Xinje XDPPro project, PLC1: XDM-60T10 (software 3.5.3 2018-12-07)

PROGRAM Ladder

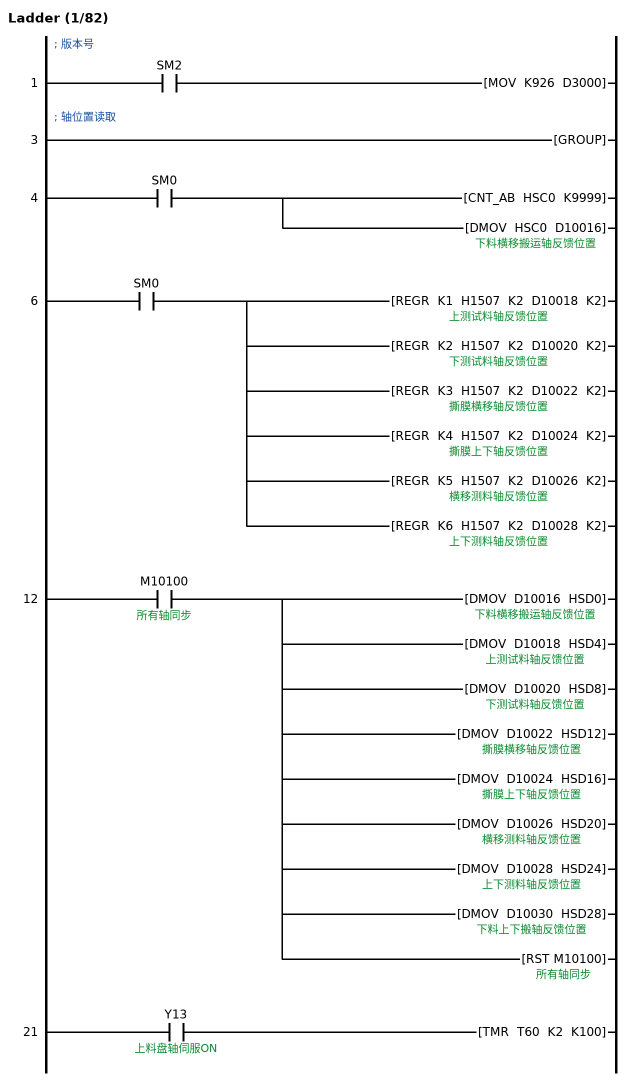
; 版本号
LD     SM2
MOV    K926 D3000
; 轴位置读取
GROUP
LD     SM0
CNT_AB HSC0 K9999
DMOV   HSC0 D10016	; 下料横移搬运轴反馈位置
LD     SM0
REGR   K1 H1507 K2 D10018 K2	; 上测试料轴反馈位置
REGR   K2 H1507 K2 D10020 K2	; 下测试料轴反馈位置
REGR   K3 H1507 K2 D10022 K2	; 撕膜横移轴反馈位置
REGR   K4 H1507 K2 D10024 K2	; 撕膜上下轴反馈位置
REGR   K5 H1507 K2 D10026 K2	; 横移测料轴反馈位置
REGR   K6 H1507 K2 D10028 K2	; 上下测料轴反馈位置
LD     M10100	; 所有轴同步
DMOV   D10016 HSD0	; 下料横移搬运轴反馈位置
DMOV   D10018 HSD4	; 上测试料轴反馈位置
DMOV   D10020 HSD8	; 下测试料轴反馈位置
DMOV   D10022 HSD12	; 撕膜横移轴反馈位置
DMOV   D10024 HSD16	; 撕膜上下轴反馈位置
DMOV   D10026 HSD20	; 横移测料轴反馈位置
DMOV   D10028 HSD24	; 上下测料轴反馈位置
DMOV   D10030 HSD28	; 下料上下搬轴反馈位置
RST    M10100	; 所有轴同步
LD     Y13	; 上料盘轴伺服ON
TMR    T60 K2 K100

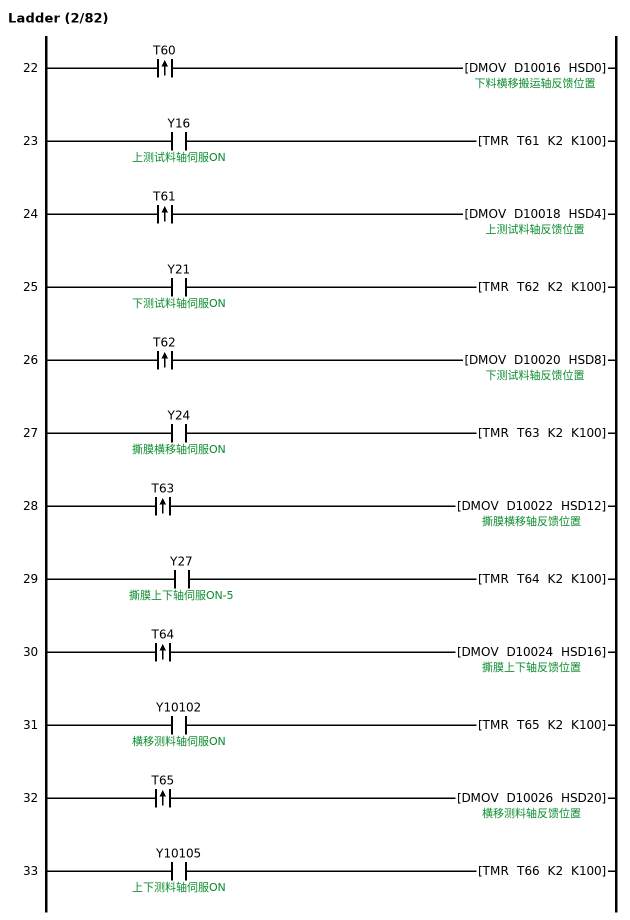
LDP    T60
DMOV   D10016 HSD0	; 下料横移搬运轴反馈位置
LD     Y16	; 上测试料轴伺服ON
TMR    T61 K2 K100
LDP    T61
DMOV   D10018 HSD4	; 上测试料轴反馈位置
LD     Y21	; 下测试料轴伺服ON
TMR    T62 K2 K100
LDP    T62
DMOV   D10020 HSD8	; 下测试料轴反馈位置
LD     Y24	; 撕膜横移轴伺服ON
TMR    T63 K2 K100
LDP    T63
DMOV   D10022 HSD12	; 撕膜横移轴反馈位置
LD     Y27	; 撕膜上下轴伺服ON-5
TMR    T64 K2 K100
LDP    T64
DMOV   D10024 HSD16	; 撕膜上下轴反馈位置
LD     Y10102	; 横移测料轴伺服ON
TMR    T65 K2 K100
LDP    T65
DMOV   D10026 HSD20	; 横移测料轴反馈位置
LD     Y10105	; 上下测料轴伺服ON
TMR    T66 K2 K100

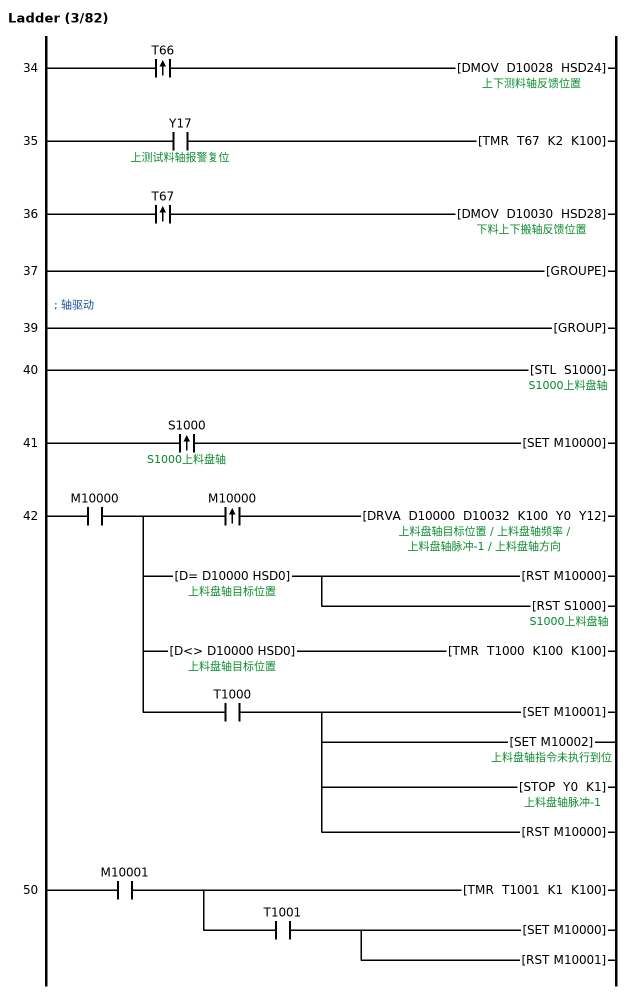
LDP    T66
DMOV   D10028 HSD24	; 上下测料轴反馈位置
LD     Y17	; 上测试料轴报警复位
TMR    T67 K2 K100
LDP    T67
DMOV   D10030 HSD28	; 下料上下搬轴反馈位置
GROUPE
; 轴驱动
GROUP
STL    S1000	; S1000上料盘轴
LDP    S1000	; S1000上料盘轴
SET    M10000
LD     M10000
MPS
ANDP   M10000
DRVA   D10000 D10032 K100 Y0 Y12	; 上料盘轴目标位置 / 上料盘轴频率 / 上料盘轴脉冲-1 / 上料盘轴方向
MRD
DAND=  D10000 HSD0	; 上料盘轴目标位置
RST    M10000
RST    S1000	; S1000上料盘轴
MRD
DAND<> D10000 HSD0	; 上料盘轴目标位置
TMR    T1000 K100 K100
MPP
AND    T1000
SET    M10001
SET    M10002	; 上料盘轴指令未执行到位
STOP   Y0 K1	; 上料盘轴脉冲-1
RST    M10000
LD     M10001
TMR    T1001 K1 K100
AND    T1001
SET    M10000
RST    M10001

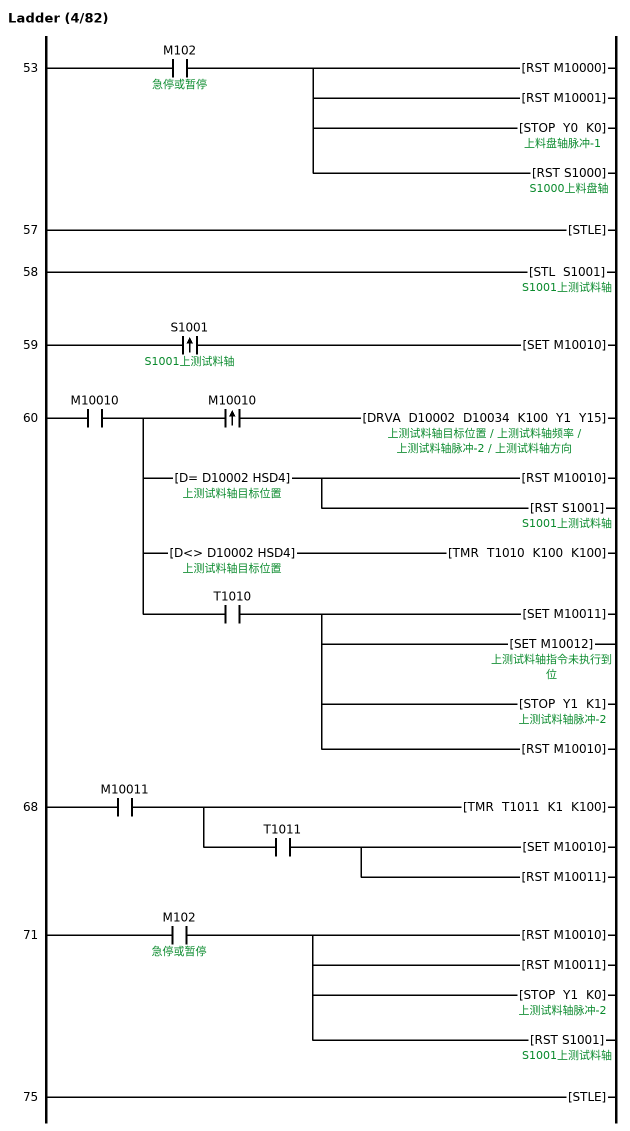
LD     M102	; 急停或暂停
RST    M10000
RST    M10001
STOP   Y0 K0	; 上料盘轴脉冲-1
RST    S1000	; S1000上料盘轴
STLE
STL    S1001	; S1001上测试料轴
LDP    S1001	; S1001上测试料轴
SET    M10010
LD     M10010
MPS
ANDP   M10010
DRVA   D10002 D10034 K100 Y1 Y15	; 上测试料轴目标位置 / 上测试料轴频率 / 上测试料轴脉冲-2 / 上测试料轴方向
MRD
DAND=  D10002 HSD4	; 上测试料轴目标位置
RST    M10010
RST    S1001	; S1001上测试料轴
MRD
DAND<> D10002 HSD4	; 上测试料轴目标位置
TMR    T1010 K100 K100
MPP
AND    T1010
SET    M10011
SET    M10012	; 上测试料轴指令未执行到位
STOP   Y1 K1	; 上测试料轴脉冲-2
RST    M10010
LD     M10011
TMR    T1011 K1 K100
AND    T1011
SET    M10010
RST    M10011
LD     M102	; 急停或暂停
RST    M10010
RST    M10011
STOP   Y1 K0	; 上测试料轴脉冲-2
RST    S1001	; S1001上测试料轴
STLE

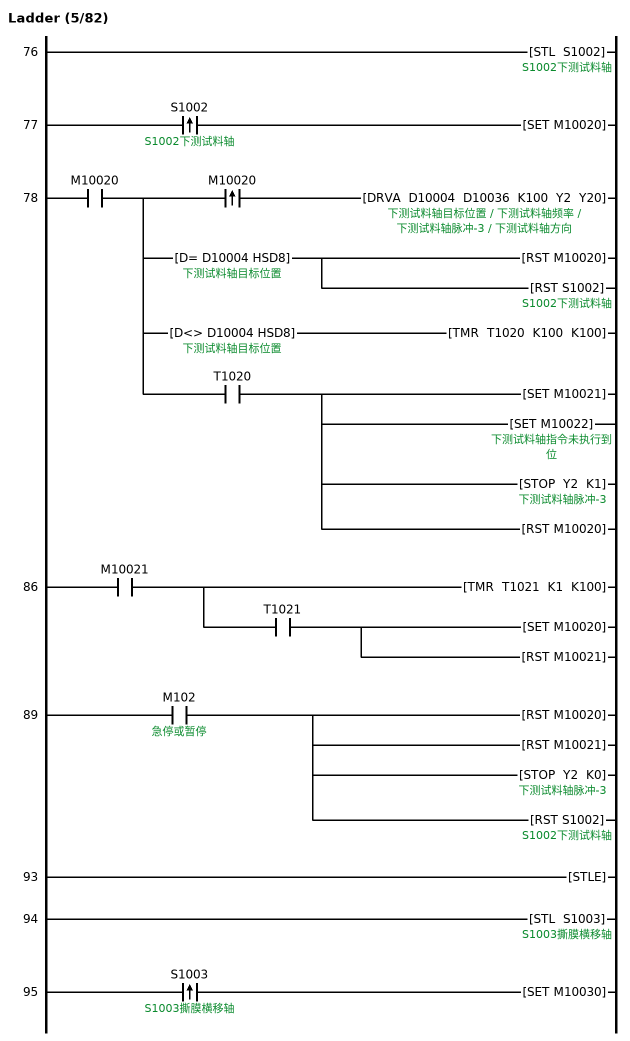
STL    S1002	; S1002下测试料轴
LDP    S1002	; S1002下测试料轴
SET    M10020
LD     M10020
MPS
ANDP   M10020
DRVA   D10004 D10036 K100 Y2 Y20	; 下测试料轴目标位置 / 下测试料轴频率 / 下测试料轴脉冲-3 / 下测试料轴方向
MRD
DAND=  D10004 HSD8	; 下测试料轴目标位置
RST    M10020
RST    S1002	; S1002下测试料轴
MRD
DAND<> D10004 HSD8	; 下测试料轴目标位置
TMR    T1020 K100 K100
MPP
AND    T1020
SET    M10021
SET    M10022	; 下测试料轴指令未执行到位
STOP   Y2 K1	; 下测试料轴脉冲-3
RST    M10020
LD     M10021
TMR    T1021 K1 K100
AND    T1021
SET    M10020
RST    M10021
LD     M102	; 急停或暂停
RST    M10020
RST    M10021
STOP   Y2 K0	; 下测试料轴脉冲-3
RST    S1002	; S1002下测试料轴
STLE
STL    S1003	; S1003撕膜横移轴
LDP    S1003	; S1003撕膜横移轴
SET    M10030

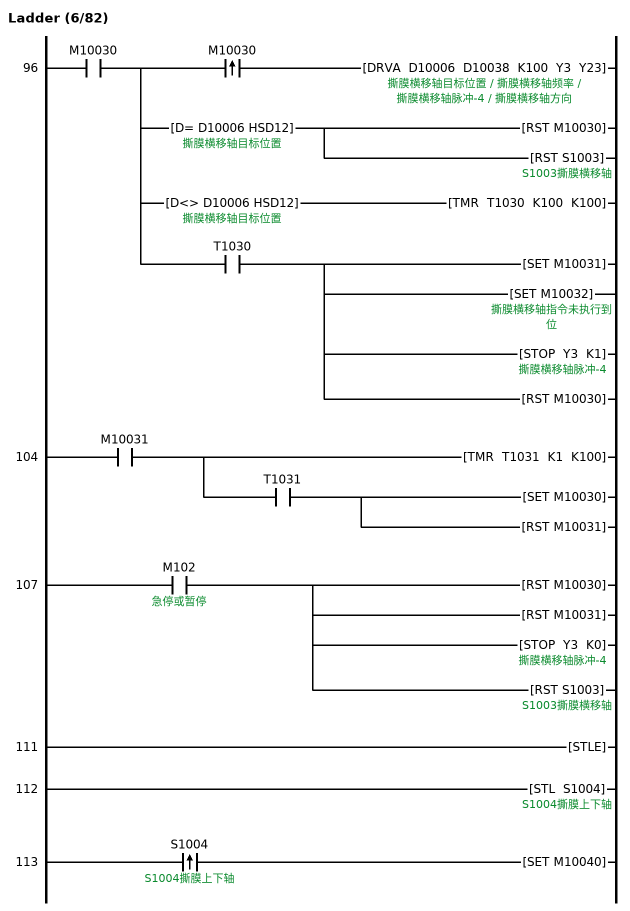
LD     M10030
MPS
ANDP   M10030
DRVA   D10006 D10038 K100 Y3 Y23	; 撕膜横移轴目标位置 / 撕膜横移轴频率 / 撕膜横移轴脉冲-4 / 撕膜横移轴方向
MRD
DAND=  D10006 HSD12	; 撕膜横移轴目标位置
RST    M10030
RST    S1003	; S1003撕膜横移轴
MRD
DAND<> D10006 HSD12	; 撕膜横移轴目标位置
TMR    T1030 K100 K100
MPP
AND    T1030
SET    M10031
SET    M10032	; 撕膜横移轴指令未执行到位
STOP   Y3 K1	; 撕膜横移轴脉冲-4
RST    M10030
LD     M10031
TMR    T1031 K1 K100
AND    T1031
SET    M10030
RST    M10031
LD     M102	; 急停或暂停
RST    M10030
RST    M10031
STOP   Y3 K0	; 撕膜横移轴脉冲-4
RST    S1003	; S1003撕膜横移轴
STLE
STL    S1004	; S1004撕膜上下轴
LDP    S1004	; S1004撕膜上下轴
SET    M10040

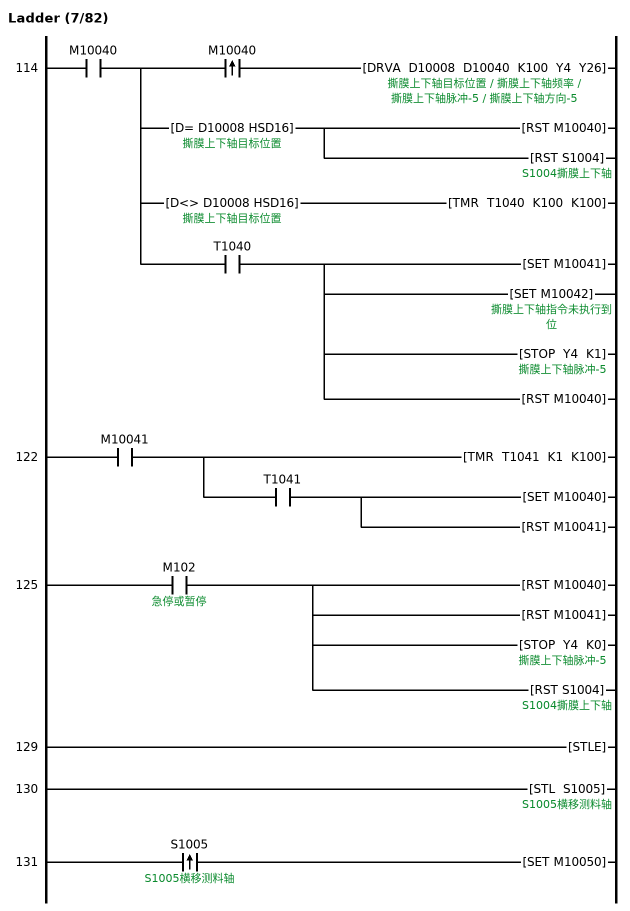
LD     M10040
MPS
ANDP   M10040
DRVA   D10008 D10040 K100 Y4 Y26	; 撕膜上下轴目标位置 / 撕膜上下轴频率 / 撕膜上下轴脉冲-5 / 撕膜上下轴方向-5
MRD
DAND=  D10008 HSD16	; 撕膜上下轴目标位置
RST    M10040
RST    S1004	; S1004撕膜上下轴
MRD
DAND<> D10008 HSD16	; 撕膜上下轴目标位置
TMR    T1040 K100 K100
MPP
AND    T1040
SET    M10041
SET    M10042	; 撕膜上下轴指令未执行到位
STOP   Y4 K1	; 撕膜上下轴脉冲-5
RST    M10040
LD     M10041
TMR    T1041 K1 K100
AND    T1041
SET    M10040
RST    M10041
LD     M102	; 急停或暂停
RST    M10040
RST    M10041
STOP   Y4 K0	; 撕膜上下轴脉冲-5
RST    S1004	; S1004撕膜上下轴
STLE
STL    S1005	; S1005横移测料轴
LDP    S1005	; S1005横移测料轴
SET    M10050

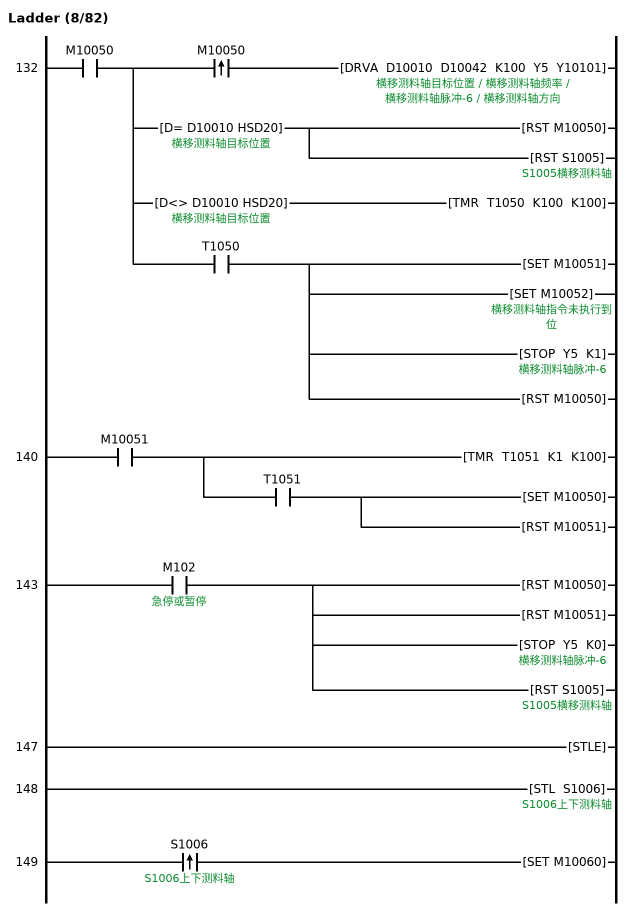
LD     M10050
MPS
ANDP   M10050
DRVA   D10010 D10042 K100 Y5 Y10101	; 横移测料轴目标位置 / 横移测料轴频率 / 横移测料轴脉冲-6 / 横移测料轴方向
MRD
DAND=  D10010 HSD20	; 横移测料轴目标位置
RST    M10050
RST    S1005	; S1005横移测料轴
MRD
DAND<> D10010 HSD20	; 横移测料轴目标位置
TMR    T1050 K100 K100
MPP
AND    T1050
SET    M10051
SET    M10052	; 横移测料轴指令未执行到位
STOP   Y5 K1	; 横移测料轴脉冲-6
RST    M10050
LD     M10051
TMR    T1051 K1 K100
AND    T1051
SET    M10050
RST    M10051
LD     M102	; 急停或暂停
RST    M10050
RST    M10051
STOP   Y5 K0	; 横移测料轴脉冲-6
RST    S1005	; S1005横移测料轴
STLE
STL    S1006	; S1006上下测料轴
LDP    S1006	; S1006上下测料轴
SET    M10060

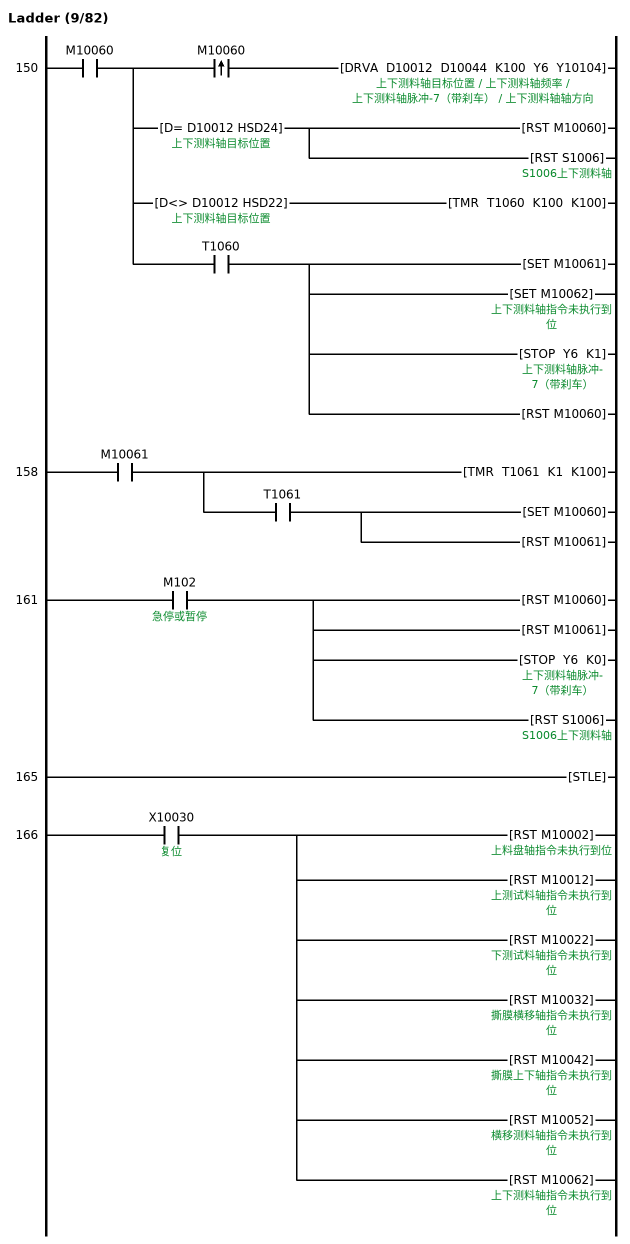
LD     M10060
MPS
ANDP   M10060
DRVA   D10012 D10044 K100 Y6 Y10104	; 上下测料轴目标位置 / 上下测料轴频率 / 上下测料轴脉冲-7（带刹车） / 上下测料轴轴方向
MRD
DAND=  D10012 HSD24	; 上下测料轴目标位置
RST    M10060
RST    S1006	; S1006上下测料轴
MRD
DAND<> D10012 HSD22	; 上下测料轴目标位置
TMR    T1060 K100 K100
MPP
AND    T1060
SET    M10061
SET    M10062	; 上下测料轴指令未执行到位
STOP   Y6 K1	; 上下测料轴脉冲-7（带刹车）
RST    M10060
LD     M10061
TMR    T1061 K1 K100
AND    T1061
SET    M10060
RST    M10061
LD     M102	; 急停或暂停
RST    M10060
RST    M10061
STOP   Y6 K0	; 上下测料轴脉冲-7（带刹车）
RST    S1006	; S1006上下测料轴
STLE
LD     X10030	; 复位
RST    M10002	; 上料盘轴指令未执行到位
RST    M10012	; 上测试料轴指令未执行到位
RST    M10022	; 下测试料轴指令未执行到位
RST    M10032	; 撕膜横移轴指令未执行到位
RST    M10042	; 撕膜上下轴指令未执行到位
RST    M10052	; 横移测料轴指令未执行到位
RST    M10062	; 上下测料轴指令未执行到位

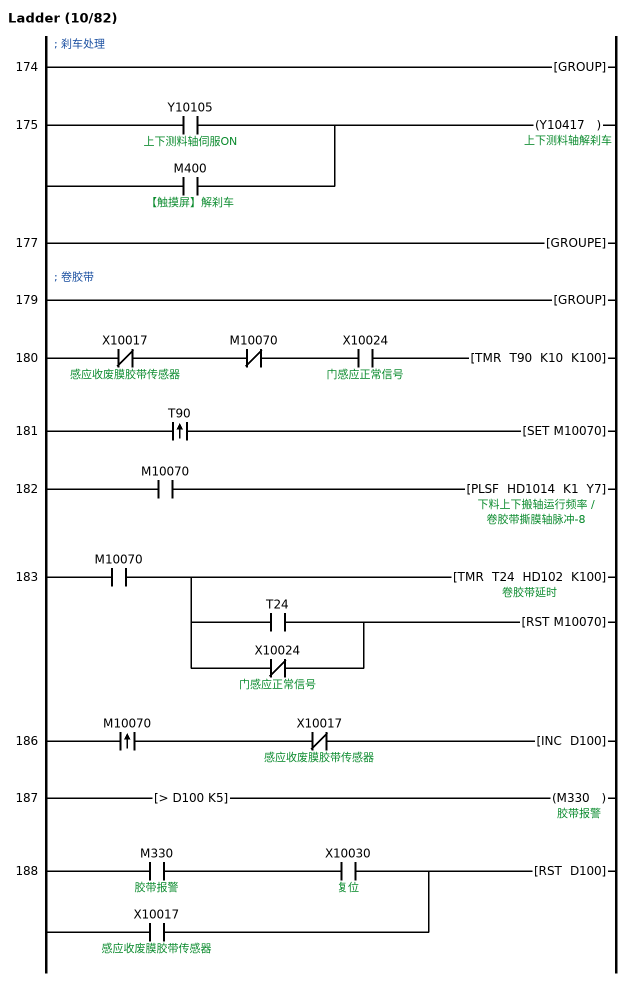
; 刹车处理
GROUP
LD     Y10105	; 上下测料轴伺服ON
OR     M400	; 【触摸屏】解刹车
OUT    Y10417	; 上下测料轴解刹车
GROUPE
; 卷胶带
GROUP
LDI    X10017	; 感应收废膜胶带传感器
ANI    M10070
AND    X10024	; 门感应正常信号
TMR    T90 K10 K100
LDP    T90
SET    M10070
LD     M10070
PLSF   HD1014 K1 Y7	; 下料上下搬轴运行频率 / 卷胶带撕膜轴脉冲-8
LD     M10070
TMR    T24 HD102 K100	; 卷胶带延时
LD     T24
ORI    X10024	; 门感应正常信号
ANB
RST    M10070
LDP    M10070
ANI    X10017	; 感应收废膜胶带传感器
INC    D100
LD>    D100 K5
OUT    M330	; 胶带报警
LD     M330	; 胶带报警
AND    X10030	; 复位
OR     X10017	; 感应收废膜胶带传感器
RST    D100

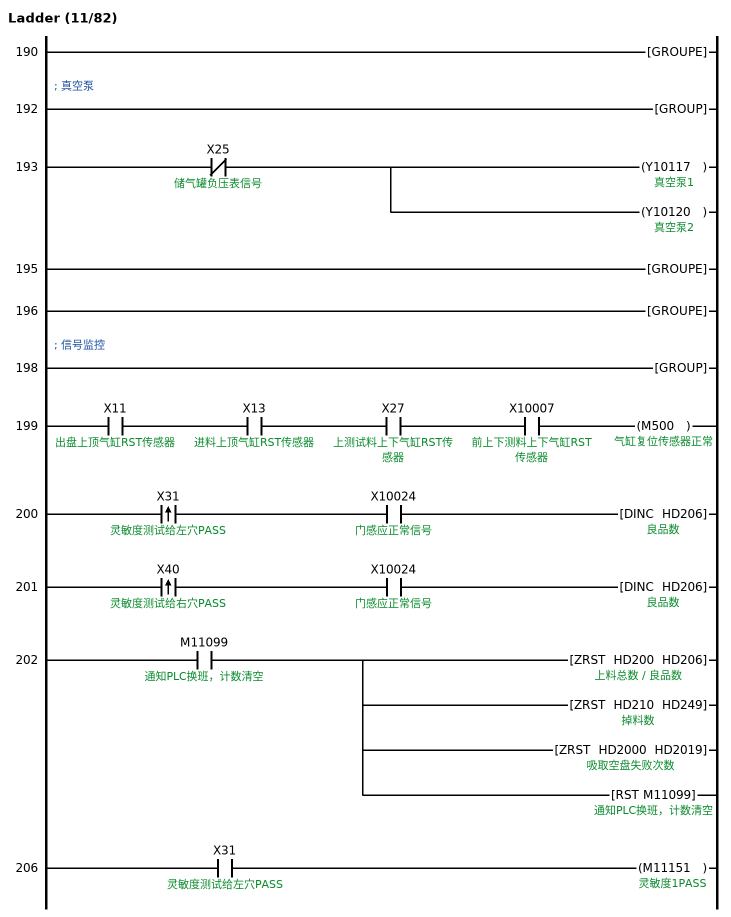
GROUPE
; 真空泵
GROUP
LDI    X25	; 储气罐负压表信号
OUT    Y10117	; 真空泵1
OUT    Y10120	; 真空泵2
GROUPE
GROUPE
; 信号监控
GROUP
LD     X11	; 出盘上顶气缸RST传感器
AND    X13	; 进料上顶气缸RST传感器
AND    X27	; 上测试料上下气缸RST传感器
AND    X10007	; 前上下测料上下气缸RST传感器
OUT    M500	; 气缸复位传感器正常
LDP    X31	; 灵敏度测试给左穴PASS
AND    X10024	; 门感应正常信号
DINC   HD206	; 良品数
LDP    X40	; 灵敏度测试给右穴PASS
AND    X10024	; 门感应正常信号
DINC   HD206	; 良品数
LD     M11099	; 通知PLC换班，计数清空
ZRST   HD200 HD206	; 上料总数 / 良品数
ZRST   HD210 HD249	; 掉料数
ZRST   HD2000 HD2019	; 吸取空盘失败次数
RST    M11099	; 通知PLC换班，计数清空
LD     X31	; 灵敏度测试给左穴PASS
OUT    M11151	; 灵敏度1PASS

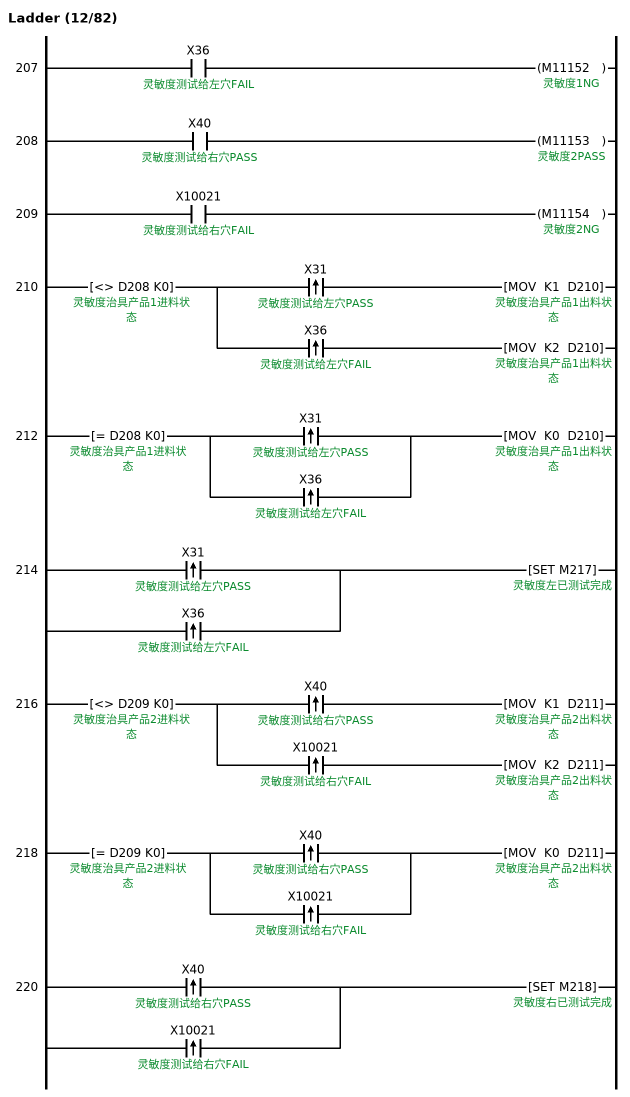
LD     X36	; 灵敏度测试给左穴FAIL
OUT    M11152	; 灵敏度1NG
LD     X40	; 灵敏度测试给右穴PASS
OUT    M11153	; 灵敏度2PASS
LD     X10021	; 灵敏度测试给右穴FAIL
OUT    M11154	; 灵敏度2NG
LD<>   D208 K0	; 灵敏度治具产品1进料状态
MPS
ANDP   X31	; 灵敏度测试给左穴PASS
MOV    K1 D210	; 灵敏度治具产品1出料状态
MPP
ANDP   X36	; 灵敏度测试给左穴FAIL
MOV    K2 D210	; 灵敏度治具产品1出料状态
LD=    D208 K0	; 灵敏度治具产品1进料状态
LDP    X31	; 灵敏度测试给左穴PASS
ORP    X36	; 灵敏度测试给左穴FAIL
ANB
MOV    K0 D210	; 灵敏度治具产品1出料状态
LDP    X31	; 灵敏度测试给左穴PASS
ORP    X36	; 灵敏度测试给左穴FAIL
SET    M217	; 灵敏度左已测试完成
LD<>   D209 K0	; 灵敏度治具产品2进料状态
MPS
ANDP   X40	; 灵敏度测试给右穴PASS
MOV    K1 D211	; 灵敏度治具产品2出料状态
MPP
ANDP   X10021	; 灵敏度测试给右穴FAIL
MOV    K2 D211	; 灵敏度治具产品2出料状态
LD=    D209 K0	; 灵敏度治具产品2进料状态
LDP    X40	; 灵敏度测试给右穴PASS
ORP    X10021	; 灵敏度测试给右穴FAIL
ANB
MOV    K0 D211	; 灵敏度治具产品2出料状态
LDP    X40	; 灵敏度测试给右穴PASS
ORP    X10021	; 灵敏度测试给右穴FAIL
SET    M218	; 灵敏度右已测试完成

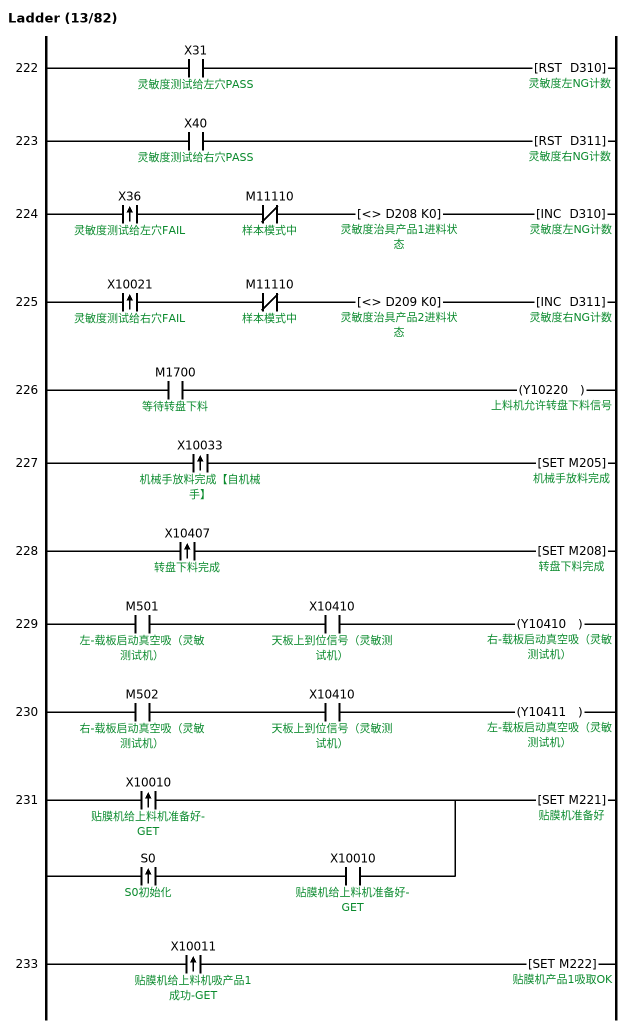
LD     X31	; 灵敏度测试给左穴PASS
RST    D310	; 灵敏度左NG计数
LD     X40	; 灵敏度测试给右穴PASS
RST    D311	; 灵敏度右NG计数
LDP    X36	; 灵敏度测试给左穴FAIL
ANI    M11110	; 样本模式中
AND<>  D208 K0	; 灵敏度治具产品1进料状态
INC    D310	; 灵敏度左NG计数
LDP    X10021	; 灵敏度测试给右穴FAIL
ANI    M11110	; 样本模式中
AND<>  D209 K0	; 灵敏度治具产品2进料状态
INC    D311	; 灵敏度右NG计数
LD     M1700	; 等待转盘下料
OUT    Y10220	; 上料机允许转盘下料信号
LDP    X10033	; 机械手放料完成【自机械手】
SET    M205	; 机械手放料完成
LDP    X10407	; 转盘下料完成
SET    M208	; 转盘下料完成
LD     M501	; 左-载板启动真空吸（灵敏测试机）
AND    X10410	; 天板上到位信号（灵敏测试机）
OUT    Y10410	; 右-载板启动真空吸（灵敏测试机）
LD     M502	; 右-载板启动真空吸（灵敏测试机）
AND    X10410	; 天板上到位信号（灵敏测试机）
OUT    Y10411	; 左-载板启动真空吸（灵敏测试机）
LDP    X10010	; 贴膜机给上料机准备好-GET
LDP    S0	; S0初始化
AND    X10010	; 贴膜机给上料机准备好-GET
ORB
SET    M221	; 贴膜机准备好
LDP    X10011	; 贴膜机给上料机吸产品1成功-GET
SET    M222	; 贴膜机产品1吸取OK

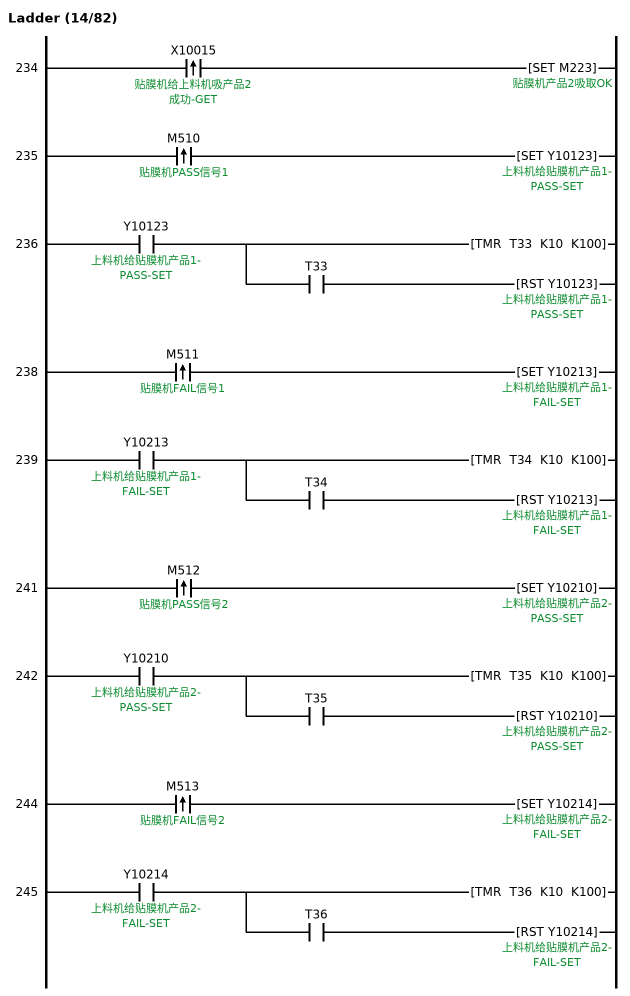
LDP    X10015	; 贴膜机给上料机吸产品2成功-GET
SET    M223	; 贴膜机产品2吸取OK
LDP    M510	; 贴膜机PASS信号1
SET    Y10123	; 上料机给贴膜机产品1-PASS-SET
LD     Y10123	; 上料机给贴膜机产品1-PASS-SET
TMR    T33 K10 K100
AND    T33
RST    Y10123	; 上料机给贴膜机产品1-PASS-SET
LDP    M511	; 贴膜机FAIL信号1
SET    Y10213	; 上料机给贴膜机产品1-FAIL-SET
LD     Y10213	; 上料机给贴膜机产品1-FAIL-SET
TMR    T34 K10 K100
AND    T34
RST    Y10213	; 上料机给贴膜机产品1-FAIL-SET
LDP    M512	; 贴膜机PASS信号2
SET    Y10210	; 上料机给贴膜机产品2-PASS-SET
LD     Y10210	; 上料机给贴膜机产品2-PASS-SET
TMR    T35 K10 K100
AND    T35
RST    Y10210	; 上料机给贴膜机产品2-PASS-SET
LDP    M513	; 贴膜机FAIL信号2
SET    Y10214	; 上料机给贴膜机产品2-FAIL-SET
LD     Y10214	; 上料机给贴膜机产品2-FAIL-SET
TMR    T36 K10 K100
AND    T36
RST    Y10214	; 上料机给贴膜机产品2-FAIL-SET

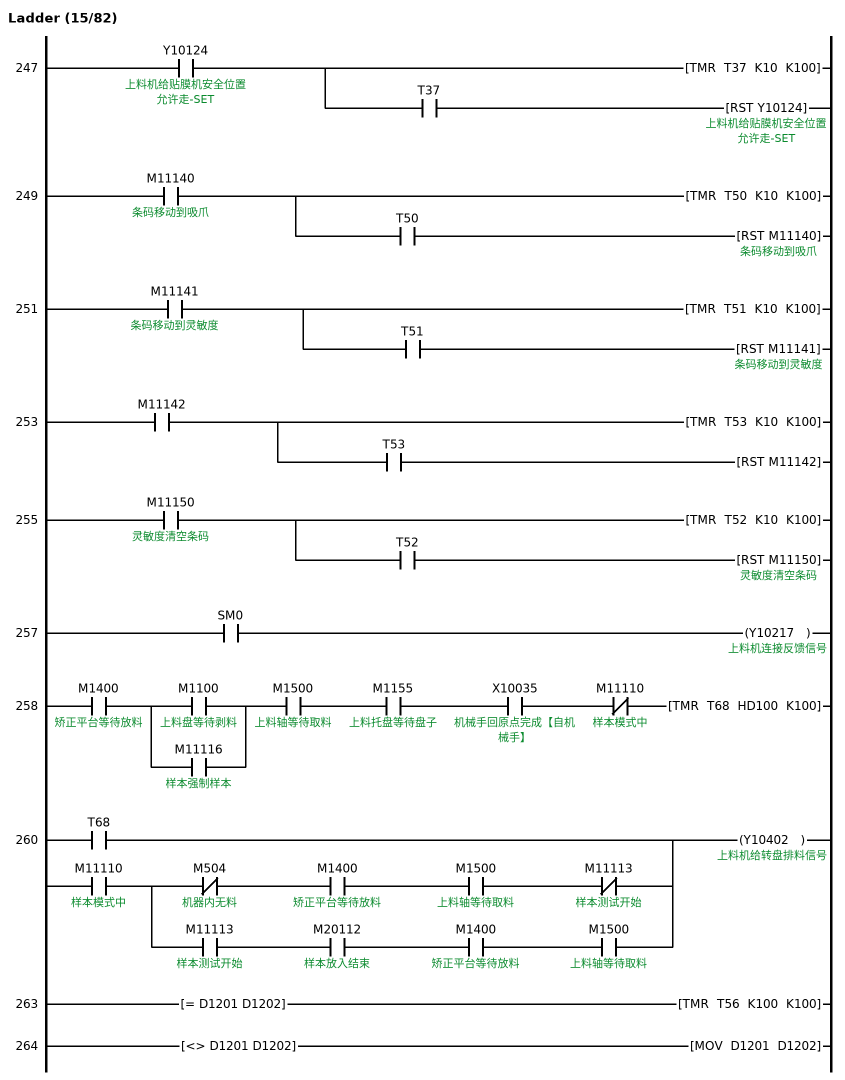
LD     Y10124	; 上料机给贴膜机安全位置允许走-SET
TMR    T37 K10 K100
AND    T37
RST    Y10124	; 上料机给贴膜机安全位置允许走-SET
LD     M11140	; 条码移动到吸爪
TMR    T50 K10 K100
AND    T50
RST    M11140	; 条码移动到吸爪
LD     M11141	; 条码移动到灵敏度
TMR    T51 K10 K100
AND    T51
RST    M11141	; 条码移动到灵敏度
LD     M11142
TMR    T53 K10 K100
AND    T53
RST    M11142
LD     M11150	; 灵敏度清空条码
TMR    T52 K10 K100
AND    T52
RST    M11150	; 灵敏度清空条码
LD     SM0
OUT    Y10217	; 上料机连接反馈信号
LD     M1400	; 矫正平台等待放料
LD     M1100	; 上料盘等待剥料
OR     M11116	; 样本强制样本
ANB
AND    M1500	; 上料轴等待取料
AND    M1155	; 上料托盘等待盘子
AND    X10035	; 机械手回原点完成【自机械手】
ANI    M11110	; 样本模式中
TMR    T68 HD100 K100
LD     T68
LD     M11110	; 样本模式中
LDI    M504	; 机器内无料
AND    M1400	; 矫正平台等待放料
AND    M1500	; 上料轴等待取料
ANI    M11113	; 样本测试开始
LD     M11113	; 样本测试开始
AND    M20112	; 样本放入结束
AND    M1400	; 矫正平台等待放料
AND    M1500	; 上料轴等待取料
ORB
ANB
ORB
OUT    Y10402	; 上料机给转盘排料信号
LD=    D1201 D1202
TMR    T56 K100 K100
LD<>   D1201 D1202
MOV    D1201 D1202

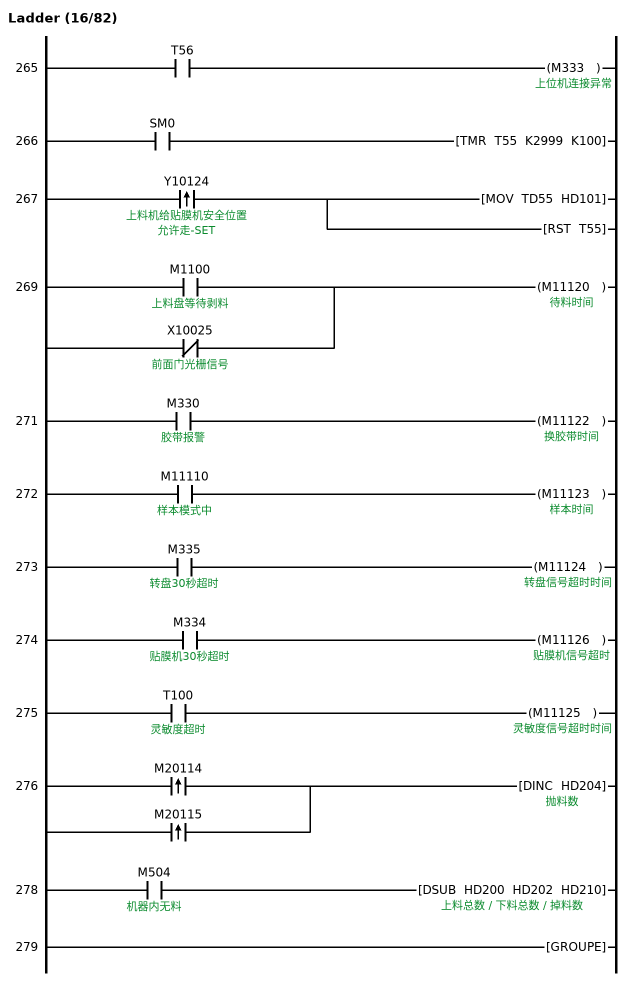
LD     T56
OUT    M333	; 上位机连接异常
LD     SM0
TMR    T55 K2999 K100
LDP    Y10124	; 上料机给贴膜机安全位置允许走-SET
MOV    TD55 HD101
RST    T55
LD     M1100	; 上料盘等待剥料
ORI    X10025	; 前面门光栅信号
OUT    M11120	; 待料时间
LD     M330	; 胶带报警
OUT    M11122	; 换胶带时间
LD     M11110	; 样本模式中
OUT    M11123	; 样本时间
LD     M335	; 转盘30秒超时
OUT    M11124	; 转盘信号超时时间
LD     M334	; 贴膜机30秒超时
OUT    M11126	; 贴膜机信号超时
LD     T100	; 灵敏度超时
OUT    M11125	; 灵敏度信号超时时间
LDP    M20114
ORP    M20115
DINC   HD204	; 抛料数
LD     M504	; 机器内无料
DSUB   HD200 HD202 HD210	; 上料总数 / 下料总数 / 掉料数
GROUPE

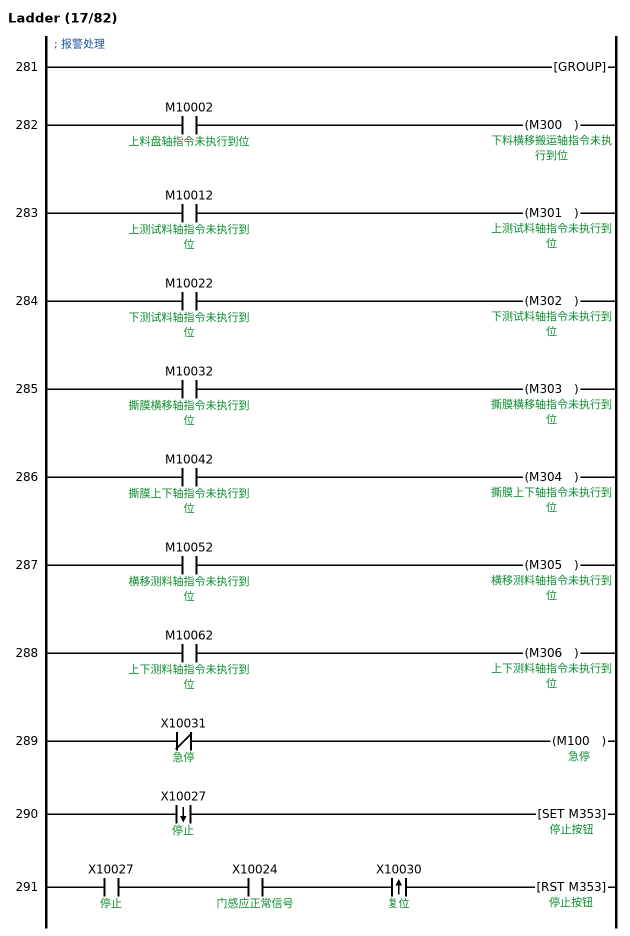
; 报警处理
GROUP
LD     M10002	; 上料盘轴指令未执行到位
OUT    M300	; 下料横移搬运轴指令未执行到位
LD     M10012	; 上测试料轴指令未执行到位
OUT    M301	; 上测试料轴指令未执行到位
LD     M10022	; 下测试料轴指令未执行到位
OUT    M302	; 下测试料轴指令未执行到位
LD     M10032	; 撕膜横移轴指令未执行到位
OUT    M303	; 撕膜横移轴指令未执行到位
LD     M10042	; 撕膜上下轴指令未执行到位
OUT    M304	; 撕膜上下轴指令未执行到位
LD     M10052	; 横移测料轴指令未执行到位
OUT    M305	; 横移测料轴指令未执行到位
LD     M10062	; 上下测料轴指令未执行到位
OUT    M306	; 上下测料轴指令未执行到位
LDI    X10031	; 急停
OUT    M100	; 急停
LDF    X10027	; 停止
SET    M353	; 停止按钮
LD     X10027	; 停止
AND    X10024	; 门感应正常信号
ANDP   X10030	; 复位
RST    M353	; 停止按钮

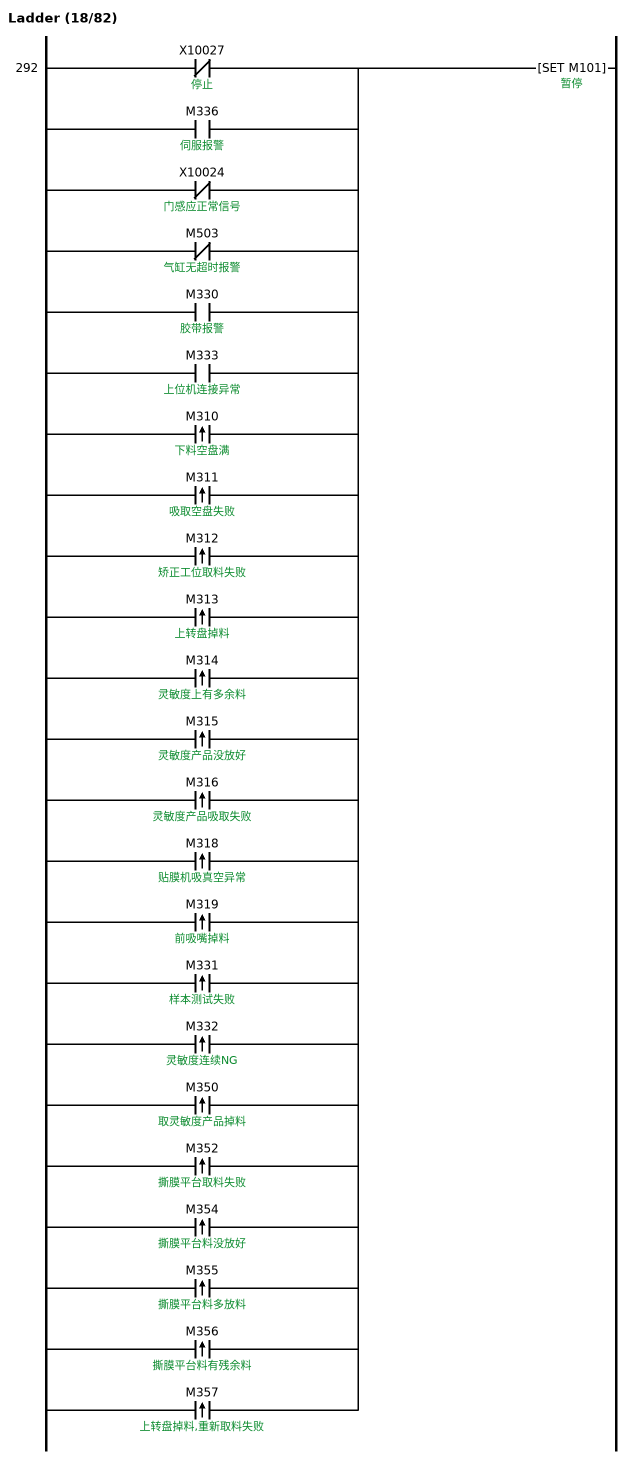
LDI    X10027	; 停止
OR     M336	; 伺服报警
ORI    X10024	; 门感应正常信号
ORI    M503	; 气缸无超时报警
OR     M330	; 胶带报警
OR     M333	; 上位机连接异常
ORP    M310	; 下料空盘满
ORP    M311	; 吸取空盘失败
ORP    M312	; 矫正工位取料失败
ORP    M313	; 上转盘掉料
ORP    M314	; 灵敏度上有多余料
ORP    M315	; 灵敏度产品没放好
ORP    M316	; 灵敏度产品吸取失败
ORP    M318	; 贴膜机吸真空异常
ORP    M319	; 前吸嘴掉料
ORP    M331	; 样本测试失败
ORP    M332	; 灵敏度连续NG
ORP    M350	; 取灵敏度产品掉料
ORP    M352	; 撕膜平台取料失败
ORP    M354	; 撕膜平台料没放好
ORP    M355	; 撕膜平台料多放料
ORP    M356	; 撕膜平台料有残余料
ORP    M357	; 上转盘掉料,重新取料失败
SET    M101	; 暂停

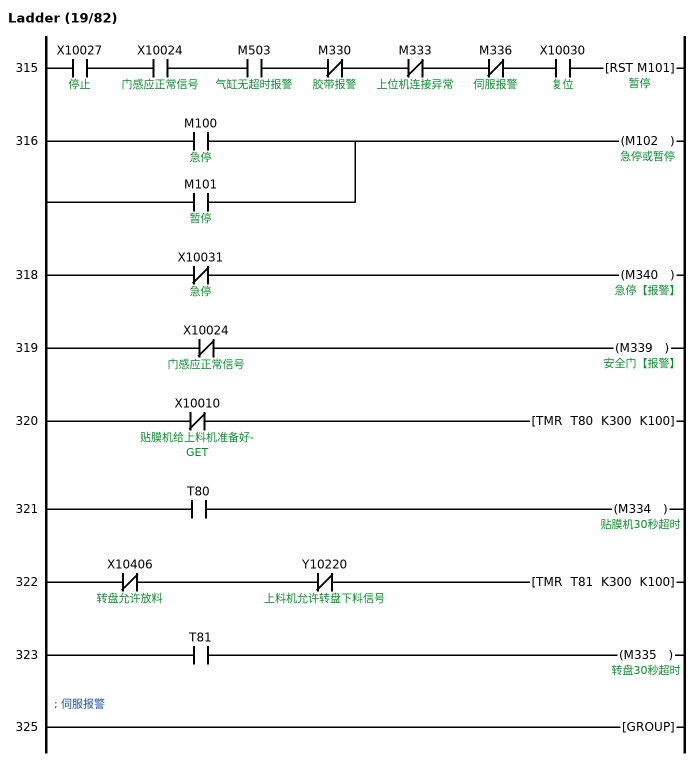
LD     X10027	; 停止
AND    X10024	; 门感应正常信号
AND    M503	; 气缸无超时报警
ANI    M330	; 胶带报警
ANI    M333	; 上位机连接异常
ANI    M336	; 伺服报警
AND    X10030	; 复位
RST    M101	; 暂停
LD     M100	; 急停
OR     M101	; 暂停
OUT    M102	; 急停或暂停
LDI    X10031	; 急停
OUT    M340	; 急停【报警】
LDI    X10024	; 门感应正常信号
OUT    M339	; 安全门【报警】
LDI    X10010	; 贴膜机给上料机准备好-GET
TMR    T80 K300 K100
LD     T80
OUT    M334	; 贴膜机30秒超时
LDI    X10406	; 转盘允许放料
ANI    Y10220	; 上料机允许转盘下料信号
TMR    T81 K300 K100
LD     T81
OUT    M335	; 转盘30秒超时
; 伺服报警
GROUP

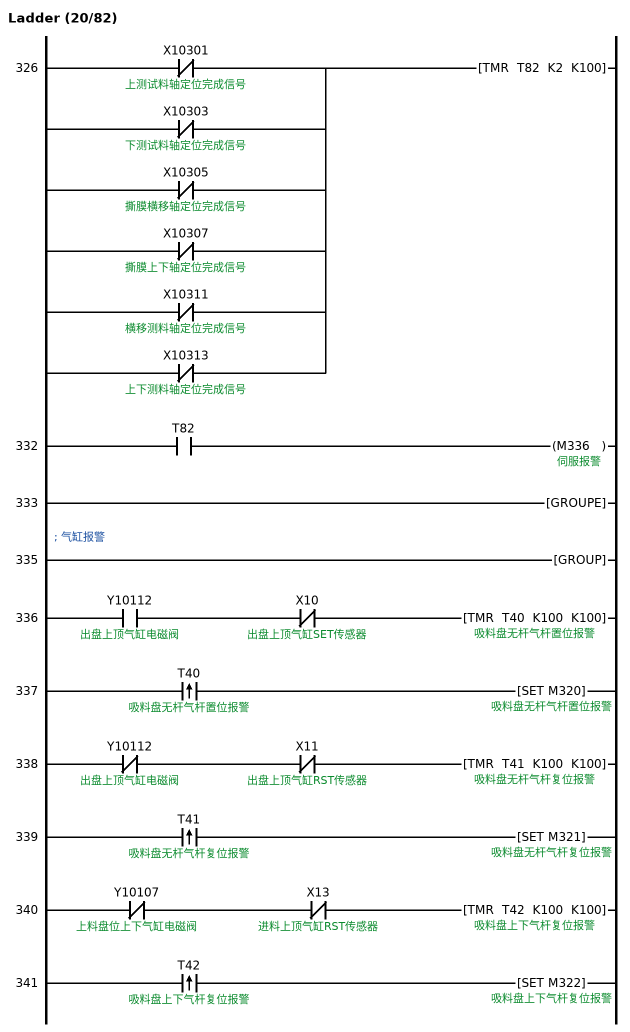
LDI    X10301	; 上测试料轴定位完成信号
ORI    X10303	; 下测试料轴定位完成信号
ORI    X10305	; 撕膜横移轴定位完成信号
ORI    X10307	; 撕膜上下轴定位完成信号
ORI    X10311	; 横移测料轴定位完成信号
ORI    X10313	; 上下测料轴定位完成信号
TMR    T82 K2 K100
LD     T82
OUT    M336	; 伺服报警
GROUPE
; 气缸报警
GROUP
LD     Y10112	; 出盘上顶气缸电磁阀
ANI    X10	; 出盘上顶气缸SET传感器
TMR    T40 K100 K100	; 吸料盘无杆气杆置位报警
LDP    T40	; 吸料盘无杆气杆置位报警
SET    M320	; 吸料盘无杆气杆置位报警
LDI    Y10112	; 出盘上顶气缸电磁阀
ANI    X11	; 出盘上顶气缸RST传感器
TMR    T41 K100 K100	; 吸料盘无杆气杆复位报警
LDP    T41	; 吸料盘无杆气杆复位报警
SET    M321	; 吸料盘无杆气杆复位报警
LDI    Y10107	; 上料盘位上下气缸电磁阀
ANI    X13	; 进料上顶气缸RST传感器
TMR    T42 K100 K100	; 吸料盘上下气杆复位报警
LDP    T42	; 吸料盘上下气杆复位报警
SET    M322	; 吸料盘上下气杆复位报警

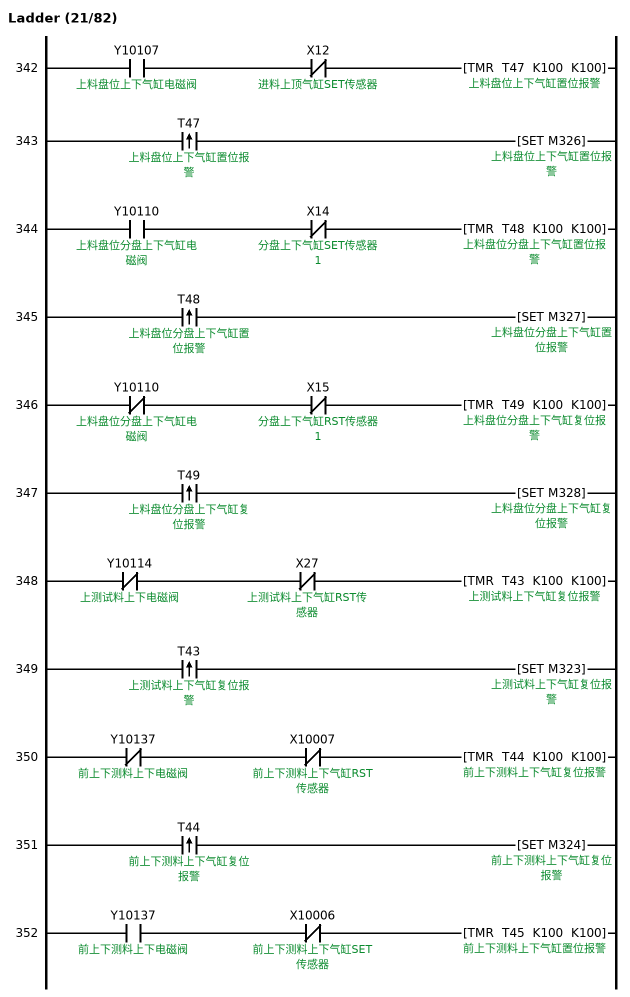
LD     Y10107	; 上料盘位上下气缸电磁阀
ANI    X12	; 进料上顶气缸SET传感器
TMR    T47 K100 K100	; 上料盘位上下气缸置位报警
LDP    T47	; 上料盘位上下气缸置位报警
SET    M326	; 上料盘位上下气缸置位报警
LD     Y10110	; 上料盘位分盘上下气缸电磁阀
ANI    X14	; 分盘上下气缸SET传感器1
TMR    T48 K100 K100	; 上料盘位分盘上下气缸置位报警
LDP    T48	; 上料盘位分盘上下气缸置位报警
SET    M327	; 上料盘位分盘上下气缸置位报警
LDI    Y10110	; 上料盘位分盘上下气缸电磁阀
ANI    X15	; 分盘上下气缸RST传感器1
TMR    T49 K100 K100	; 上料盘位分盘上下气缸复位报警
LDP    T49	; 上料盘位分盘上下气缸复位报警
SET    M328	; 上料盘位分盘上下气缸复位报警
LDI    Y10114	; 上测试料上下电磁阀
ANI    X27	; 上测试料上下气缸RST传感器
TMR    T43 K100 K100	; 上测试料上下气缸复位报警
LDP    T43	; 上测试料上下气缸复位报警
SET    M323	; 上测试料上下气缸复位报警
LDI    Y10137	; 前上下测料上下电磁阀
ANI    X10007	; 前上下测料上下气缸RST传感器
TMR    T44 K100 K100	; 前上下测料上下气缸复位报警
LDP    T44	; 前上下测料上下气缸复位报警
SET    M324	; 前上下测料上下气缸复位报警
LD     Y10137	; 前上下测料上下电磁阀
ANI    X10006	; 前上下测料上下气缸SET传感器
TMR    T45 K100 K100	; 前上下测料上下气缸置位报警

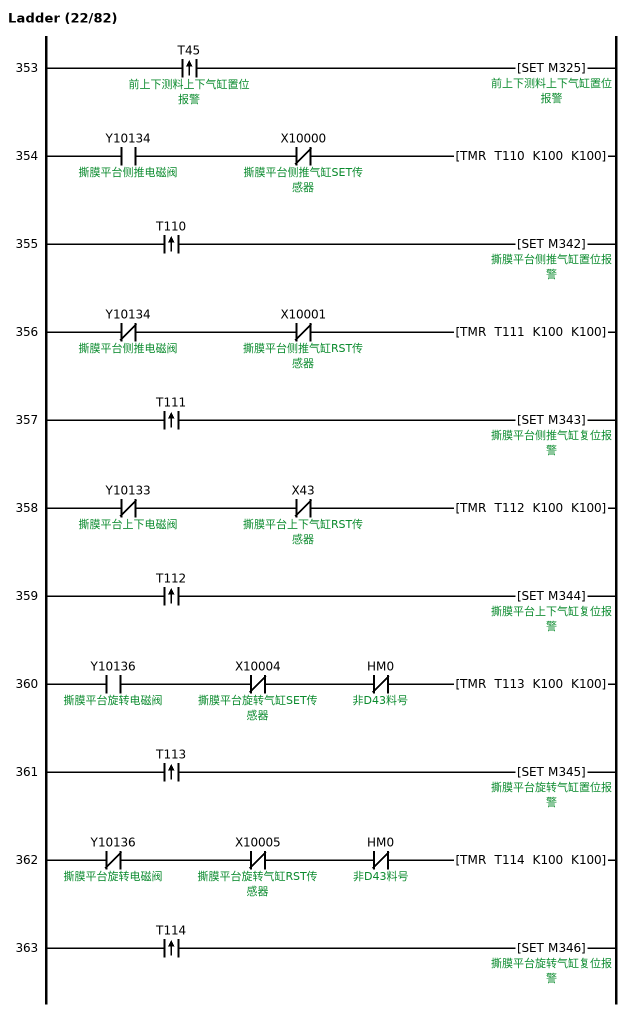
LDP    T45	; 前上下测料上下气缸置位报警
SET    M325	; 前上下测料上下气缸置位报警
LD     Y10134	; 撕膜平台侧推电磁阀
ANI    X10000	; 撕膜平台侧推气缸SET传感器
TMR    T110 K100 K100
LDP    T110
SET    M342	; 撕膜平台侧推气缸置位报警
LDI    Y10134	; 撕膜平台侧推电磁阀
ANI    X10001	; 撕膜平台侧推气缸RST传感器
TMR    T111 K100 K100
LDP    T111
SET    M343	; 撕膜平台侧推气缸复位报警
LDI    Y10133	; 撕膜平台上下电磁阀
ANI    X43	; 撕膜平台上下气缸RST传感器
TMR    T112 K100 K100
LDP    T112
SET    M344	; 撕膜平台上下气缸复位报警
LD     Y10136	; 撕膜平台旋转电磁阀
ANI    X10004	; 撕膜平台旋转气缸SET传感器
ANI    HM0	; 非D43料号
TMR    T113 K100 K100
LDP    T113
SET    M345	; 撕膜平台旋转气缸置位报警
LDI    Y10136	; 撕膜平台旋转电磁阀
ANI    X10005	; 撕膜平台旋转气缸RST传感器
ANI    HM0	; 非D43料号
TMR    T114 K100 K100
LDP    T114
SET    M346	; 撕膜平台旋转气缸复位报警

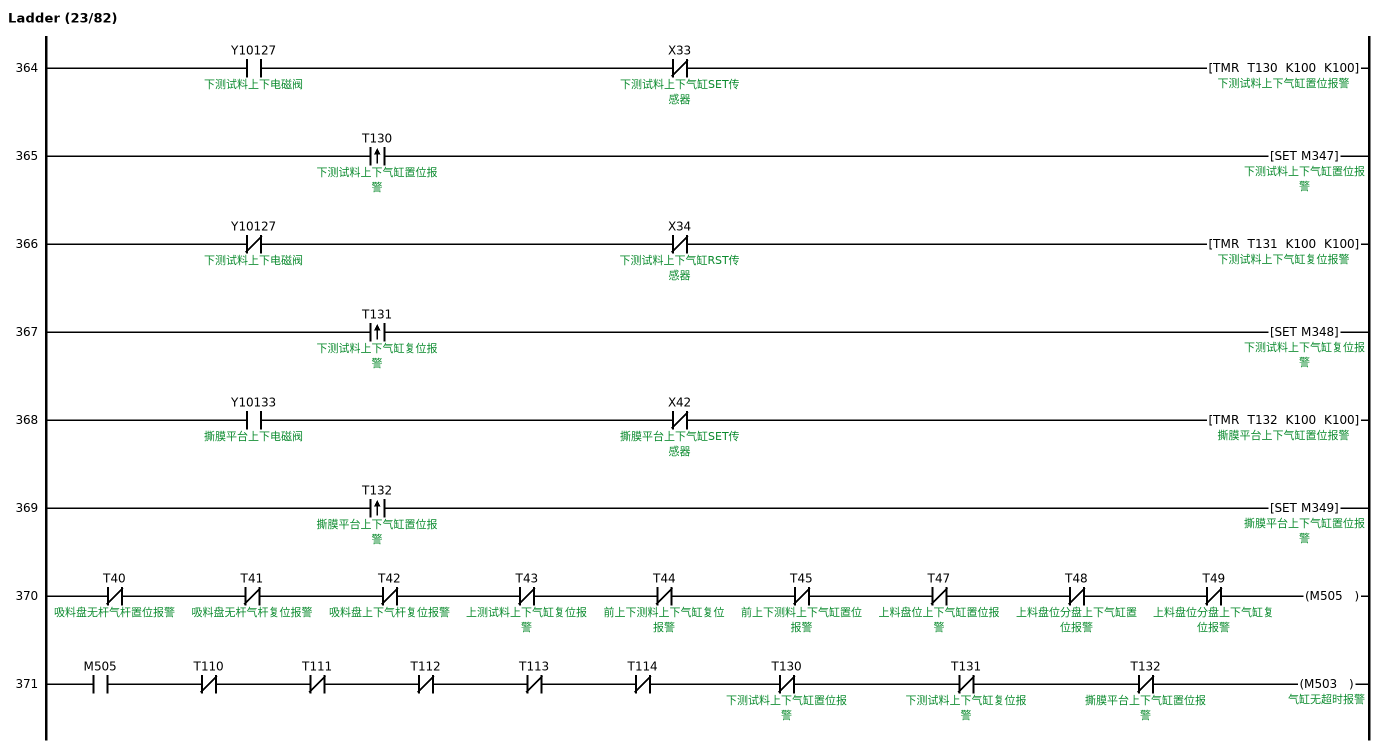
LD     Y10127	; 下测试料上下电磁阀
ANI    X33	; 下测试料上下气缸SET传感器
TMR    T130 K100 K100	; 下测试料上下气缸置位报警
LDP    T130	; 下测试料上下气缸置位报警
SET    M347	; 下测试料上下气缸置位报警
LDI    Y10127	; 下测试料上下电磁阀
ANI    X34	; 下测试料上下气缸RST传感器
TMR    T131 K100 K100	; 下测试料上下气缸复位报警
LDP    T131	; 下测试料上下气缸复位报警
SET    M348	; 下测试料上下气缸复位报警
LD     Y10133	; 撕膜平台上下电磁阀
ANI    X42	; 撕膜平台上下气缸SET传感器
TMR    T132 K100 K100	; 撕膜平台上下气缸置位报警
LDP    T132	; 撕膜平台上下气缸置位报警
SET    M349	; 撕膜平台上下气缸置位报警
LDI    T40	; 吸料盘无杆气杆置位报警
ANI    T41	; 吸料盘无杆气杆复位报警
ANI    T42	; 吸料盘上下气杆复位报警
ANI    T43	; 上测试料上下气缸复位报警
ANI    T44	; 前上下测料上下气缸复位报警
ANI    T45	; 前上下测料上下气缸置位报警
ANI    T47	; 上料盘位上下气缸置位报警
ANI    T48	; 上料盘位分盘上下气缸置位报警
ANI    T49	; 上料盘位分盘上下气缸复位报警
OUT    M505
LD     M505
ANI    T110
ANI    T111
ANI    T112
ANI    T113
ANI    T114
ANI    T130	; 下测试料上下气缸置位报警
ANI    T131	; 下测试料上下气缸复位报警
ANI    T132	; 撕膜平台上下气缸置位报警
OUT    M503	; 气缸无超时报警

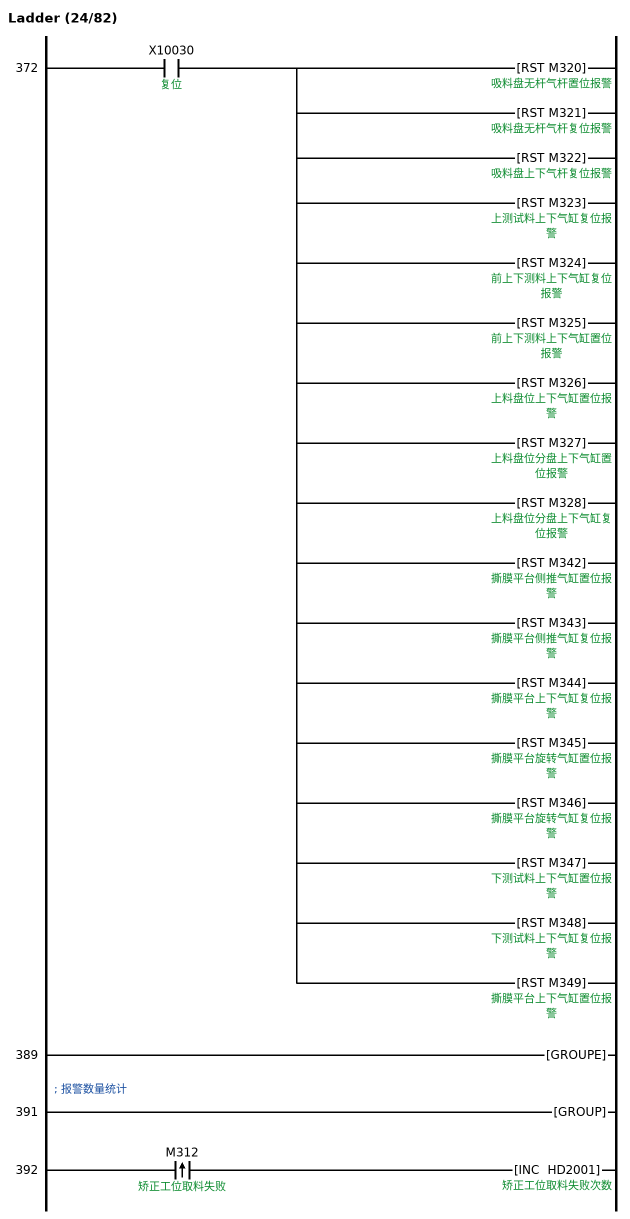
LD     X10030	; 复位
RST    M320	; 吸料盘无杆气杆置位报警
RST    M321	; 吸料盘无杆气杆复位报警
RST    M322	; 吸料盘上下气杆复位报警
RST    M323	; 上测试料上下气缸复位报警
RST    M324	; 前上下测料上下气缸复位报警
RST    M325	; 前上下测料上下气缸置位报警
RST    M326	; 上料盘位上下气缸置位报警
RST    M327	; 上料盘位分盘上下气缸置位报警
RST    M328	; 上料盘位分盘上下气缸复位报警
RST    M342	; 撕膜平台侧推气缸置位报警
RST    M343	; 撕膜平台侧推气缸复位报警
RST    M344	; 撕膜平台上下气缸复位报警
RST    M345	; 撕膜平台旋转气缸置位报警
RST    M346	; 撕膜平台旋转气缸复位报警
RST    M347	; 下测试料上下气缸置位报警
RST    M348	; 下测试料上下气缸复位报警
RST    M349	; 撕膜平台上下气缸置位报警
GROUPE
; 报警数量统计
GROUP
LDP    M312	; 矫正工位取料失败
INC    HD2001	; 矫正工位取料失败次数

